PROGRAM MP_3_Y102
VAR
	CompareOutput102_00: CMP_OC_DW;
	CompareOutput102_01: CMP_OC_DW;
	CompareOutput102_02: CMP_OC_DW;
	CompareOutput102_03: CMP_OC_DW;
	CompareOutput102_04: CMP_OC_DW;
	CompareOutput102_05: CMP_OC_DW;
	CompareOutput102_06: CMP_OC_DW;
	CompareOutput102_07: CMP_OC_DW;
	CompareOutput102_08: CMP_OC_DW;
	CompareOutput102_09: CMP_OC_DW;
	CompareOutput102_10: CMP_OC_DW;
	CompareOutput102_11: CMP_OC_DW;
	CompareOutput102_12: CMP_OC_DW;
	CompareOutput102_13: CMP_OC_DW;
	CompareOutput102_14: CMP_OC_DW;
	CompareOutput102_15: CMP_OC_DW;
END_VAR

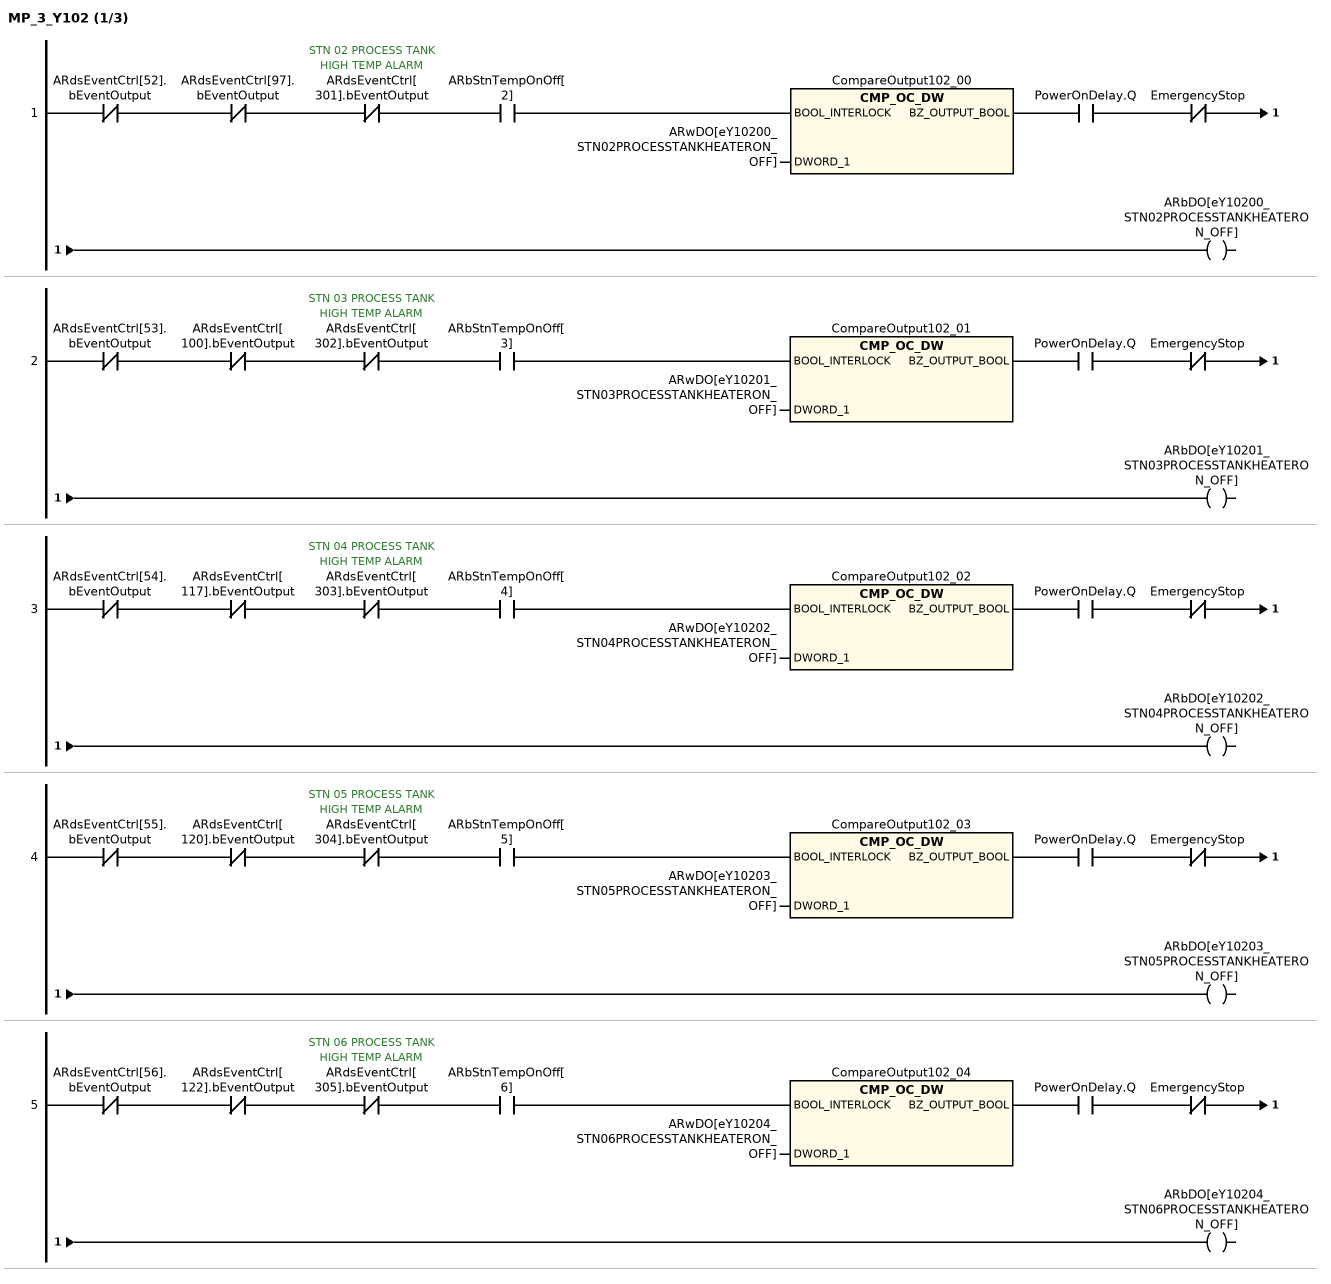
// NETWORK 1
//   ARdsEventCtrl[301].bEventOutput: STN 02 PROCESS TANK HIGH TEMP ALARM
CompareOutput102_00(BOOL_INTERLOCK := NOT ARdsEventCtrl[52].bEventOutput AND NOT ARdsEventCtrl[97].bEventOutput AND NOT ARdsEventCtrl[301].bEventOutput AND ARbStnTempOnOff[2], DWORD_1 := ARwDO[eY10200_STN02PROCESSTANKHEATERON_OFF]); // CMP_OC_DW
ARbDO[eY10200_STN02PROCESSTANKHEATERON_OFF] := CompareOutput102_00.BZ_OUTPUT_BOOL AND PowerOnDelay.Q AND NOT EmergencyStop;

// NETWORK 2
//   ARdsEventCtrl[302].bEventOutput: STN 03 PROCESS TANK HIGH TEMP ALARM
CompareOutput102_01(BOOL_INTERLOCK := NOT ARdsEventCtrl[53].bEventOutput AND NOT ARdsEventCtrl[100].bEventOutput AND NOT ARdsEventCtrl[302].bEventOutput AND ARbStnTempOnOff[3], DWORD_1 := ARwDO[eY10201_STN03PROCESSTANKHEATERON_OFF]); // CMP_OC_DW
ARbDO[eY10201_STN03PROCESSTANKHEATERON_OFF] := CompareOutput102_01.BZ_OUTPUT_BOOL AND PowerOnDelay.Q AND NOT EmergencyStop;

// NETWORK 3
//   ARdsEventCtrl[303].bEventOutput: STN 04 PROCESS TANK HIGH TEMP ALARM
CompareOutput102_02(BOOL_INTERLOCK := NOT ARdsEventCtrl[54].bEventOutput AND NOT ARdsEventCtrl[117].bEventOutput AND NOT ARdsEventCtrl[303].bEventOutput AND ARbStnTempOnOff[4], DWORD_1 := ARwDO[eY10202_STN04PROCESSTANKHEATERON_OFF]); // CMP_OC_DW
ARbDO[eY10202_STN04PROCESSTANKHEATERON_OFF] := CompareOutput102_02.BZ_OUTPUT_BOOL AND PowerOnDelay.Q AND NOT EmergencyStop;

// NETWORK 4
//   ARdsEventCtrl[304].bEventOutput: STN 05 PROCESS TANK HIGH TEMP ALARM
CompareOutput102_03(BOOL_INTERLOCK := NOT ARdsEventCtrl[55].bEventOutput AND NOT ARdsEventCtrl[120].bEventOutput AND NOT ARdsEventCtrl[304].bEventOutput AND ARbStnTempOnOff[5], DWORD_1 := ARwDO[eY10203_STN05PROCESSTANKHEATERON_OFF]); // CMP_OC_DW
ARbDO[eY10203_STN05PROCESSTANKHEATERON_OFF] := CompareOutput102_03.BZ_OUTPUT_BOOL AND PowerOnDelay.Q AND NOT EmergencyStop;

// NETWORK 5
//   ARdsEventCtrl[305].bEventOutput: STN 06 PROCESS TANK HIGH TEMP ALARM
CompareOutput102_04(BOOL_INTERLOCK := NOT ARdsEventCtrl[56].bEventOutput AND NOT ARdsEventCtrl[122].bEventOutput AND NOT ARdsEventCtrl[305].bEventOutput AND ARbStnTempOnOff[6], DWORD_1 := ARwDO[eY10204_STN06PROCESSTANKHEATERON_OFF]); // CMP_OC_DW
ARbDO[eY10204_STN06PROCESSTANKHEATERON_OFF] := CompareOutput102_04.BZ_OUTPUT_BOOL AND PowerOnDelay.Q AND NOT EmergencyStop;

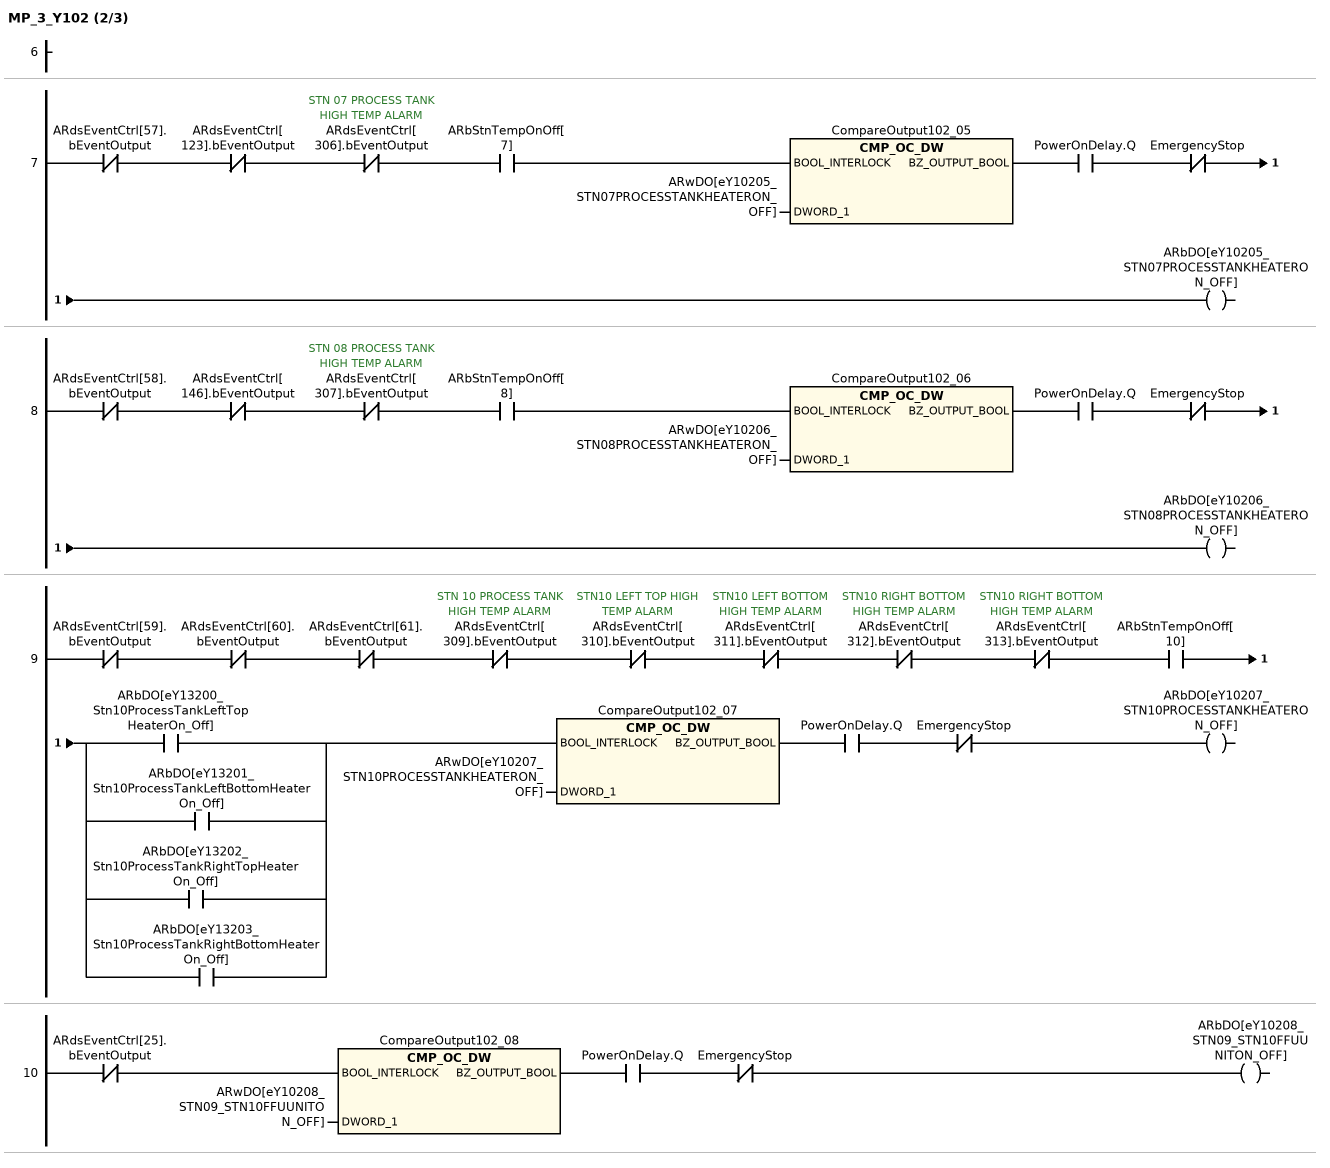
// NETWORK 6

// NETWORK 7
//   ARdsEventCtrl[306].bEventOutput: STN 07 PROCESS TANK HIGH TEMP ALARM
CompareOutput102_05(BOOL_INTERLOCK := NOT ARdsEventCtrl[57].bEventOutput AND NOT ARdsEventCtrl[123].bEventOutput AND NOT ARdsEventCtrl[306].bEventOutput AND ARbStnTempOnOff[7], DWORD_1 := ARwDO[eY10205_STN07PROCESSTANKHEATERON_OFF]); // CMP_OC_DW
ARbDO[eY10205_STN07PROCESSTANKHEATERON_OFF] := CompareOutput102_05.BZ_OUTPUT_BOOL AND PowerOnDelay.Q AND NOT EmergencyStop;

// NETWORK 8
//   ARdsEventCtrl[307].bEventOutput: STN 08 PROCESS TANK HIGH TEMP ALARM
CompareOutput102_06(BOOL_INTERLOCK := NOT ARdsEventCtrl[58].bEventOutput AND NOT ARdsEventCtrl[146].bEventOutput AND NOT ARdsEventCtrl[307].bEventOutput AND ARbStnTempOnOff[8], DWORD_1 := ARwDO[eY10206_STN08PROCESSTANKHEATERON_OFF]); // CMP_OC_DW
ARbDO[eY10206_STN08PROCESSTANKHEATERON_OFF] := CompareOutput102_06.BZ_OUTPUT_BOOL AND PowerOnDelay.Q AND NOT EmergencyStop;

// NETWORK 9
//   ARdsEventCtrl[309].bEventOutput: STN 10 PROCESS TANK HIGH TEMP ALARM
//   ARdsEventCtrl[310].bEventOutput: STN10 LEFT TOP HIGH TEMP ALARM
//   ARdsEventCtrl[311].bEventOutput: STN10 LEFT BOTTOM HIGH TEMP ALARM
//   ARdsEventCtrl[312].bEventOutput: STN10 RIGHT BOTTOM HIGH TEMP ALARM
//   ARdsEventCtrl[313].bEventOutput: STN10 RIGHT BOTTOM HIGH TEMP ALARM
CompareOutput102_07(BOOL_INTERLOCK := NOT ARdsEventCtrl[59].bEventOutput AND NOT ARdsEventCtrl[60].bEventOutput AND NOT ARdsEventCtrl[61].bEventOutput AND NOT ARdsEventCtrl[309].bEventOutput AND NOT ARdsEventCtrl[310].bEventOutput AND NOT ARdsEventCtrl[311].bEventOutput AND NOT ARdsEventCtrl[312].bEventOutput AND NOT ARdsEventCtrl[313].bEventOutput AND ARbStnTempOnOff[10] AND (ARbDO[eY13200_Stn10ProcessTankLeftTopHeaterOn_Off] OR ARbDO[eY13201_Stn10ProcessTankLeftBottomHeaterOn_Off] OR ARbDO[eY13202_Stn10ProcessTankRightTopHeaterOn_Off] OR ARbDO[eY13203_Stn10ProcessTankRightBottomHeaterOn_Off]), DWORD_1 := ARwDO[eY10207_STN10PROCESSTANKHEATERON_OFF]); // CMP_OC_DW
ARbDO[eY10207_STN10PROCESSTANKHEATERON_OFF] := CompareOutput102_07.BZ_OUTPUT_BOOL AND PowerOnDelay.Q AND NOT EmergencyStop;

// NETWORK 10
CompareOutput102_08(BOOL_INTERLOCK := NOT ARdsEventCtrl[25].bEventOutput, DWORD_1 := ARwDO[eY10208_STN09_STN10FFUUNITON_OFF]); // CMP_OC_DW
ARbDO[eY10208_STN09_STN10FFUUNITON_OFF] := CompareOutput102_08.BZ_OUTPUT_BOOL AND PowerOnDelay.Q AND NOT EmergencyStop;

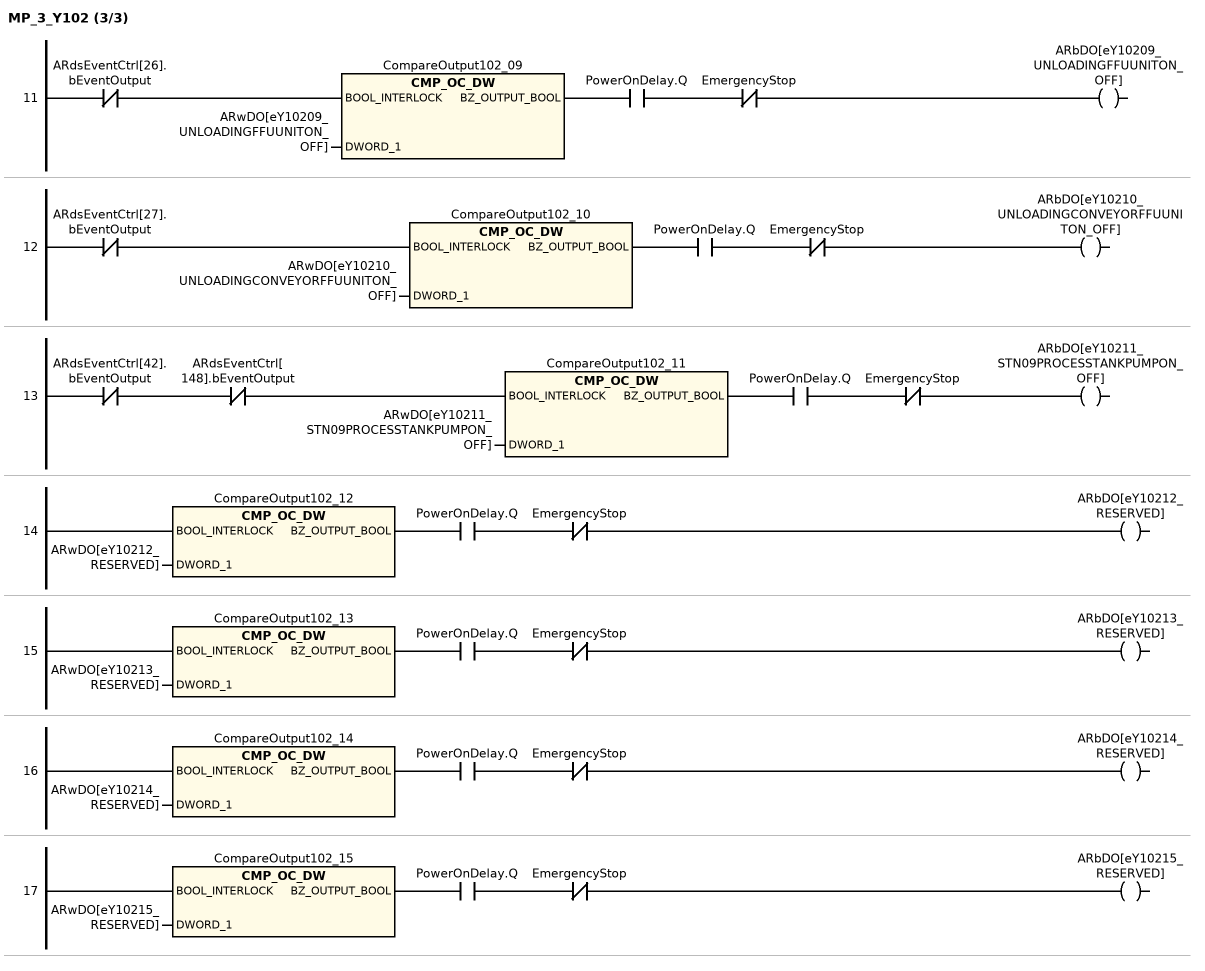
// NETWORK 11
CompareOutput102_09(BOOL_INTERLOCK := NOT ARdsEventCtrl[26].bEventOutput, DWORD_1 := ARwDO[eY10209_UNLOADINGFFUUNITON_OFF]); // CMP_OC_DW
ARbDO[eY10209_UNLOADINGFFUUNITON_OFF] := CompareOutput102_09.BZ_OUTPUT_BOOL AND PowerOnDelay.Q AND NOT EmergencyStop;

// NETWORK 12
CompareOutput102_10(BOOL_INTERLOCK := NOT ARdsEventCtrl[27].bEventOutput, DWORD_1 := ARwDO[eY10210_UNLOADINGCONVEYORFFUUNITON_OFF]); // CMP_OC_DW
ARbDO[eY10210_UNLOADINGCONVEYORFFUUNITON_OFF] := CompareOutput102_10.BZ_OUTPUT_BOOL AND PowerOnDelay.Q AND NOT EmergencyStop;

// NETWORK 13
CompareOutput102_11(BOOL_INTERLOCK := NOT ARdsEventCtrl[42].bEventOutput AND NOT ARdsEventCtrl[148].bEventOutput, DWORD_1 := ARwDO[eY10211_STN09PROCESSTANKPUMPON_OFF]); // CMP_OC_DW
ARbDO[eY10211_STN09PROCESSTANKPUMPON_OFF] := CompareOutput102_11.BZ_OUTPUT_BOOL AND PowerOnDelay.Q AND NOT EmergencyStop;

// NETWORK 14
CompareOutput102_12(BOOL_INTERLOCK := TRUE, DWORD_1 := ARwDO[eY10212_RESERVED]); // CMP_OC_DW
ARbDO[eY10212_RESERVED] := CompareOutput102_12.BZ_OUTPUT_BOOL AND PowerOnDelay.Q AND NOT EmergencyStop;

// NETWORK 15
CompareOutput102_13(BOOL_INTERLOCK := TRUE, DWORD_1 := ARwDO[eY10213_RESERVED]); // CMP_OC_DW
ARbDO[eY10213_RESERVED] := CompareOutput102_13.BZ_OUTPUT_BOOL AND PowerOnDelay.Q AND NOT EmergencyStop;

// NETWORK 16
CompareOutput102_14(BOOL_INTERLOCK := TRUE, DWORD_1 := ARwDO[eY10214_RESERVED]); // CMP_OC_DW
ARbDO[eY10214_RESERVED] := CompareOutput102_14.BZ_OUTPUT_BOOL AND PowerOnDelay.Q AND NOT EmergencyStop;

// NETWORK 17
CompareOutput102_15(BOOL_INTERLOCK := TRUE, DWORD_1 := ARwDO[eY10215_RESERVED]); // CMP_OC_DW
ARbDO[eY10215_RESERVED] := CompareOutput102_15.BZ_OUTPUT_BOOL AND PowerOnDelay.Q AND NOT EmergencyStop;

END_PROGRAM

(* stored: Version 1.1.0.1, ProductVersion 3.1.4024.11
   POU MP_3_Y102: Id {9f76dd86-8082-4df4-b1f3-56e238e4df25}, SpecialFunc None *)
